# EPICS substitutions: ek9000App/Db/EL1804.substitutions
file EL1804.template
{       pattern
        {
                TERMINAL,

        }
        {
        }
}
